FUNCTION_BLOCK FB_WareHouse EXTENDS FB_Objectbase
VAR_INPUT
	 Motors 		  : REFERENCE TO UNI_MotorList;
	 WheelhouseSensor : REFERENCE TO UNI_HMI_WheelHouseInput;
END_VAR
VAR_OUTPUT
END_VAR
VAR
   
    nMotorIndex    : UINT;
    CabinetJob     : E_CabinetJob := E_CabinetJob.Idle;    

    stLayerStatus    : st_LayerStatus;
    stWarehouseLayer : st_WarehouseLayer;
    stWarehouseList  : st_WarehouseList;
    _stWarehouseList : _st_WarehouseList;

	fbReloadBox : FB_ReloadBox;
	fbFeedInBox : FB_FeedInBox;
END_VAR

SUPER^.M_clcUpdate();
THIS^.M_clcUpdate();

PROPERTY PUBLIC bFeedInBox_Completed : BOOL
GET
bFeedInBox_Completed := fbFeedInBox.Done;
END_GET
END_PROPERTY

PROPERTY bReloadBox_Completed : BOOL
GET
bReloadBox_Completed := fbReloadBox.Done;
END_GET
END_PROPERTY

METHOD M_clcFBs : BOOL
VAR_INPUT	
END_VAR
VAR
	nELIndex			:	INT;
END_VAR
fbReloadBox(
	Execute:= , 
	Abort:= , 
	Reset:= , 
	ObjectName:= 'Warehouse Reload box', 
	Busy=> bBusy, 
	Done=> bDone, 
	Aborted=> , 
	Error=> bError, 
	ErrorID=> , 
	Status=> , 
	Motors:= Motors, 
	WarehouseStatus:= WheelhouseSensor.List,
	ArrivedDelayTime:= T#1S,
	WarehouseSelect:= ,
	WarehouseCoordinates:= , 
	TimeOut:= T#10S);
	
fbFeedInBox(
	Execute:= , 
	Abort:= , 
	Reset:= , 
	ObjectName:= 'Warehouse FeedIn box', 
	Busy=> bBusy, 
	Done=> bDone, 
	Aborted=> , 
	Error=> bError, 
	ErrorID=> , 
	Status=> , 
	Motors:= Motors, 
	WarehouseStatus:= WheelhouseSensor.List,
	ArrivedDelayTime:= T#1S,
	WarehouseSelect:= ,
	WarehouseCoordinates:= , 
	TimeOut:= T#10S);
END_METHOD

METHOD M_clcUpdate : BOOL
VAR_INPUT	
END_VAR
VAR	
	i : INT;
END_VAR
//clc FBs
M_clcFBs();
END_METHOD

METHOD PRIVATE M_GotoCommandStep : BOOL
VAR_INPUT
END_VAR
CabinetJob := E_CabinetJob.Initial;
END_METHOD

METHOD PRIVATE M_GotoErrorStep : BOOL
VAR_INPUT
END_VAR
CabinetJob := E_CabinetJob.error;
END_METHOD

METHOD PUBLIC M_ResetFeedInBox : BOOL
VAR_INPUT
END_VAR
VAR
	uiMotorInder : UINT; 
END_VAR
// reset reload box execute
fbFeedInBox.Execute := FALSE;
 
M_ResetFeedInBox := TRUE; // Method end
END_METHOD

METHOD M_ResetReloadBox : Bool
VAR_INPUT
END_VAR
// reset reload box execute
fbReloadBox.Execute := FALSE;

M_ResetReloadBox := true; // Method end
END_METHOD

METHOD PUBLIC M_StartFeedInBox : BOOL
VAR_INPUT
	WareHouseSelect : E_WareHouse;
	WarehouseCoordinates : ST_WareHouseCoordinates;
END_VAR
// Send command to Feedin box fb
fbFeedInBox.WarehouseSelect := WareHouseSelect;
fbFeedInBox.WarehouseCoordinates := WarehouseCoordinates;
fbFeedInBox.Execute := TRUE;

M_StartFeedInBox := TRUE; // Method end
END_METHOD

METHOD M_StartReloadBox : BOOL
VAR_INPUT
	WareHouseSelect : E_WareHouse;
	WarehouseCoordinates : ST_WareHouseCoordinates;
END_VAR
// Send command to reload box fb
fbReloadBox.WarehouseSelect := WareHouseSelect;
fbReloadBox.WarehouseCoordinates := WarehouseCoordinates;
fbReloadBox.Execute := TRUE;

M_StartReloadBox := true; // Method end
END_METHOD

END_FUNCTION_BLOCK

(* stored: Version 1.1.0.1, ProductVersion 3.1.4024.13
   POU FB_WareHouse: Id {9e34fd6d-a388-4d89-ad3c-398bb6e81101}, SpecialFunc None
   Folder Private: Id {db09577f-eb2b-47c1-a52b-dae3fd8202aa}
   Folder Property: Id {bb2235b2-a2c9-483d-9eb5-f9250ec26d07}
   Folder Public: Id {7decc950-39da-4c47-ba15-9910095d4e79}
   Property bFeedInBox_Completed: Id {1a121a0b-5fea-4b2f-98ce-48de81120080}
   Get Get: Id {c36db18e-453d-49fe-9631-767a2fd2c62e}
   Property bReloadBox_Completed: Id {d094b7e4-02a0-4847-8cc4-6ce221d9dfa1}
   Get Get: Id {6b3b17bf-4a42-4193-a77e-d4e5e1d85cf9}
   Method M_clcFBs: Id {807c3ae5-39b2-4244-84be-cbe713bcde55}
   Method M_clcUpdate: Id {701c4651-0044-45e4-8c49-c7027fc05428}
   Method M_GotoCommandStep: Id {70bb7f48-95b9-42f9-92fd-88a6b932af74}
   Method M_GotoErrorStep: Id {7392dba7-e112-4341-ac92-00c5c2ab3ce3}
   Method M_ResetFeedInBox: Id {2a934a59-1200-4f64-811f-54910fd6220d}
   Method M_ResetReloadBox: Id {c6c9a42a-9b24-4a85-8550-77ba05aeb881}
   Method M_StartFeedInBox: Id {96df12ea-7239-4aa6-a966-7188a4268391}
   Method M_StartReloadBox: Id {707d4576-a459-43b2-8d3a-60f9ff63aa4d} *)
